# B&R Automation Studio project trialproject1
Automation Studio 4.5.2.102

## Configuration Config1

### Task classes (Cpu.sw)
```
Cyclic#1 (cycle 2000 us, tolerance 0 us):
  ncsdcctrl <- ncsdcctrl.prg
Cyclic#4:
  Program <- Program.prg
NcDataObjects: acp10etxen <- acp10etxen.dob, gAxis01a <- gAxis01obj.gAxis01a.dob, gAxis01i <- gAxis01obj.gAxis01i.dob
VcDataObjects: Visu <- gAxis01obj.Visu.dob
Libraries: Acp10man, Acp10par, NcGlobal, Acp10sdc, AsBrStr, Acp10_MC, brsystem, sys_lib, runtime, Library
```

### Hardware
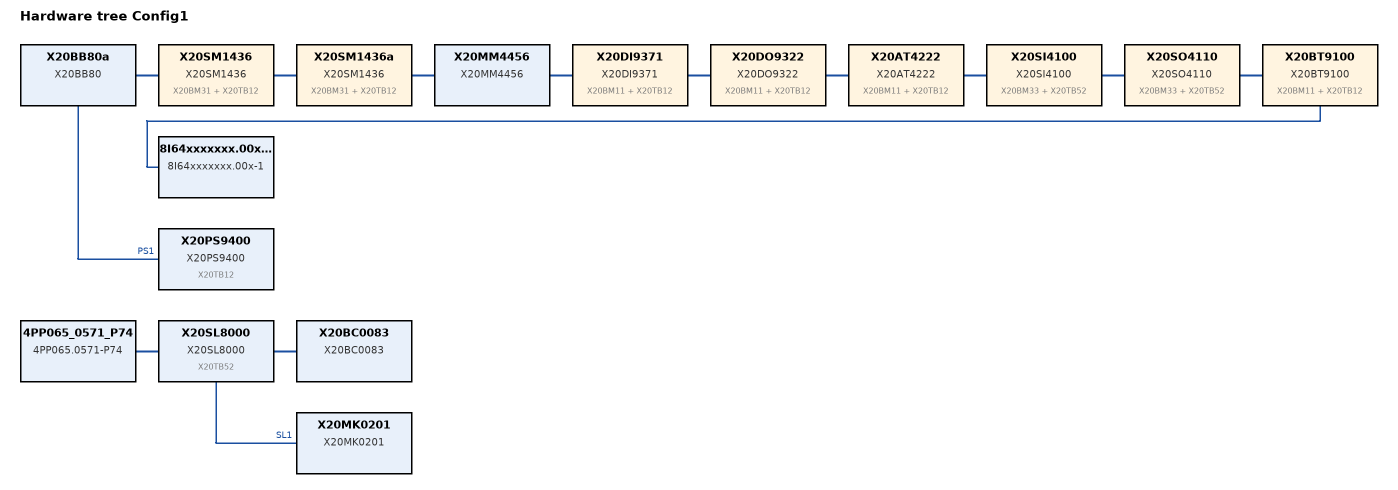
```
4PP065_0571_P74 : 4PP065.0571-P74 v1.1.2.0
  Connector IF5:
    ActivateDevice = 1
    Mode = Manual
    InternetAddress = 10.0.1.10
    SubnetMask = 255.255.255.0
  ConfigurationID = labBR
  RebootReset = 2
  TimerDeviceType = EPLX2X
  TimerDevice = 4PP065_0571_P74.IF4
  TaskClassIdleTime = 2000
  Cyclic1Duration = 2000
  Cyclic1Tolerance = 0
  Cyclic1Output = 1
  VcObjectName = Visu
8I64xxxxxxx.00x-1 : 8I64xxxxxxx.00x-1 v2.1.2.0  [X2X1 -> X20BT9100.X2X1 [Cable Type=X2XCable, Length=10, Version=1.0.0.2]]
  packedETAD = packed
  packedCMDD = packed
X20AT4222 : X20AT4222 v1.2.3.0  [SS1 -> X20TB12f.SS; SL -> X20BM11c.SL1]
X20BB80a : X20BB80 v1.0.2.0
X20BC0083 : X20BC0083 v2.7.0.0  [PLK1 -> X20SL8000.PLK2 (NodeNumber=2) [Cable Type=PowerlinkCable, Length=10, Version=1.0.0.2]; SL -> X20BB80a.SL1]
X20BM11a : X20BM11 v1.0.0.1  [X2X1 -> X20MM4456.X2X2]
X20BM11b : X20BM11 v1.0.0.1  [X2X1 -> X20BM11a.X2X2]
X20BM11c : X20BM11 v1.0.0.1  [X2X1 -> X20BM11b.X2X2]
X20BM11d : X20BM11 v1.0.0.1  [X2X1 -> X20BM33b.X2X2]
X20BM31a : X20BM31 v1.0.0.1  [X2X1 -> X20BB80a.IF1]
X20BM31b : X20BM31 v1.0.0.1  [X2X1 -> X20BM31a.X2X2]
X20BM33a : X20BM33 v1.0.0.4  [X2X1 -> X20BM11c.X2X2]
X20BM33b : X20BM33 v1.0.0.4  [X2X1 -> X20BM33a.X2X2]
X20BT9100 : X20BT9100 v1.0.3.0  [SS1 -> X20TB12g.SS; SL -> X20BM11d.SL1]
X20DI9371 : X20DI9371 v1.0.2.0  [SS1 -> X20TB12d.SS; SL -> X20BM11a.SL1]
X20DO9322 : X20DO9322 v1.0.3.0  [SS1 -> X20TB12e.SS; SL -> X20BM11b.SL1]
X20MK0201 : X20MK0201 v1.0.0.0  [SL -> X20SL8000.SL1]
X20MM4456 : X20MM4456 v1.1.5.0  [X2X1 -> X20BM31b.X2X2]
X20PS9400 : X20PS9400 v1.0.2.4  [SS1 -> X20TB12.SS; PS -> X20BB80a.PS1]
X20SI4100 : X20SI4100 v1.10.1.1  [SS1 -> X20TB52b.SS; SL -> X20BM33a.SL1]
X20SL8000 : X20SL8000 v1.6.5.1  [PLK1 -> 4PP065_0571_P74.IF4 (NodeNumber=1) [Cable Type=PowerlinkCable, Length=10, Version=1.0.0.2]; PLK2 -> X20BC0083.PLK1 (NodeNumber=1) [Cable Type=PowerlinkCable, Length=10, Version=1.0.0.2]; SS1 -> X20TB52.SS]
  SafeProject = SafeLOGIC-1
X20SM1436 : X20SM1436 v1.4.2.1  [SS1 -> X20TB12a.SS; SL -> X20BM31a.SL1]
X20SM1436a : X20SM1436 v1.4.2.1  [SS1 -> X20TB12c.SS; SL -> X20BM31b.SL1]
X20SO4110 : X20SO4110 v1.10.1.1  [SS1 -> X20TB52c.SS; SL -> X20BM33b.SL1]
  SafeModuleID = 3
X20TB12 : X20TB12 v1.0.0.0
X20TB12a : X20TB12 v1.0.0.0
X20TB12c : X20TB12 v1.0.0.0
X20TB12d : X20TB12 v1.0.0.0
X20TB12e : X20TB12 v1.0.0.0
X20TB12f : X20TB12 v1.0.0.0
X20TB12g : X20TB12 v1.0.0.0
X20TB52 : X20TB52 v1.0.0.1
X20TB52b : X20TB52 v1.0.0.1
X20TB52c : X20TB52 v1.0.0.1
```

## Logical view

### Global.var
```iecst
VAR
	gAxis01 : ACP10AXIS_typ;
	gAxis01_HW : SdcHwCfg_typ := (0);
	gAxis01_DrvIf : SdcDrvIf16_typ := (0);
	gAxis01_DiDoIf : SdcDiDoIf_typ := (0);
	gAxis01_ModuleOk : BOOL := 0;
	speed : INT := 500;
	EVIRD : DRIVE;
	start : INT := 0;
END_VAR
```

### Program Logical/Program

#### Main.c
```c
#include <bur/plctypes.h>

#ifdef _DEFAULT_INCLUDES
#include <AsDefault.h>
#endif

void _INIT ProgramInit(void)
{
	speed=500;
	EVIRD.ENABLED=1;
}

void _CYCLIC ProgramCyclic(void)
{
	DRIVE(&EVIRD);
	if(start == 0)  //Остановка двигателя если отжата кнопка Start
	{
		speed=0;
	}
}

void _EXIT ProgramExit(void)
{

}
```
